% RSLogix 500 project CTD QUE 3.RSS, saved by version 8.30.00.15 %
PROJECT "UNTITLED"    % processor: MicroLogix 1400 %

PROGRAM FILES
  LAD 2   6 rungs

DATA FILES
  O0 OUTPUT  6 elements
  I1 INPUT  8 elements
  S2 STATUS  66 elements
  B3 BINARY  1 elements
  T4 TIMER  1 elements
  C5 COUNTER  6 elements
  R6 CONTROL  1 elements
  N7 INTEGER  1 elements
  F8 FLOAT  1 elements

LADDER 2
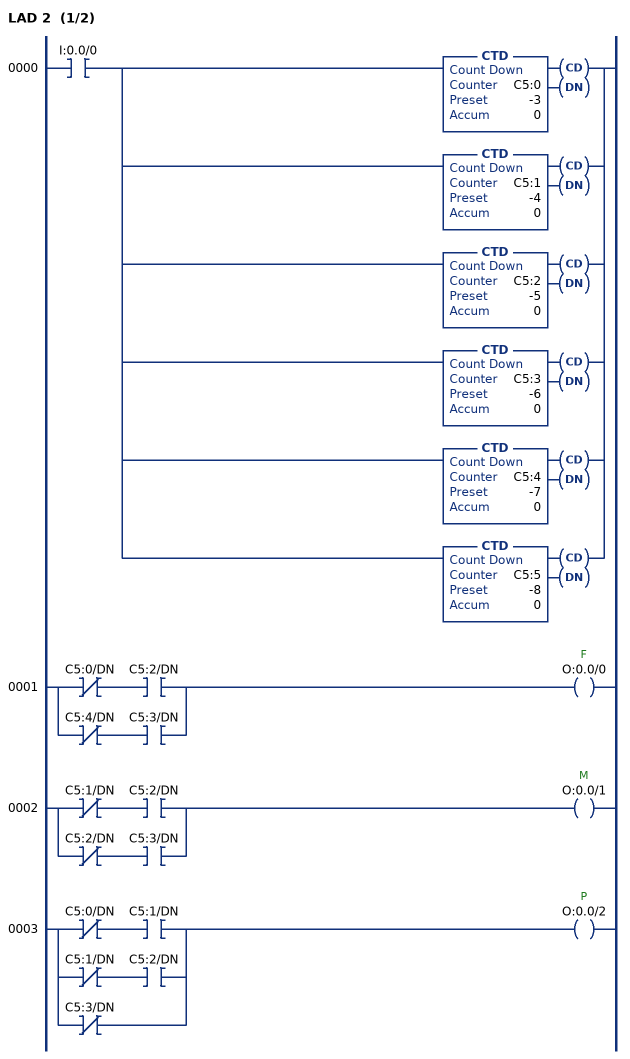
% Rung: 0 %  % edit flag set %
SOR XIC I:0.0/0 BST CTD C5:0 -3 0 NXB BST CTD C5:1 -4 0 NXB BST CTD C5:2 -5 0 NXB BST CTD C5:3 -6 0 NXB BST CTD C5:4 -7 0 NXB CTD C5:5 -8 0 BND BND BND BND BND EOR
% Rung: 1 %
SOR BST XIO C5:0/DN XIC C5:2/DN NXB XIO C5:4/DN XIC C5:3/DN BND OTE O:0.0/0 EOR
%   O:0.0/0  F %
% Rung: 2 %
SOR BST XIO C5:1/DN XIC C5:2/DN NXB XIO C5:2/DN XIC C5:3/DN BND OTE O:0.0/1 EOR
%   O:0.0/1  M %
% Rung: 3 %
SOR BST XIO C5:0/DN XIC C5:1/DN NXB BST XIO C5:1/DN XIC C5:2/DN NXB XIO C5:3/DN BND BND OTE O:0.0/2 EOR
%   O:0.0/2  P %

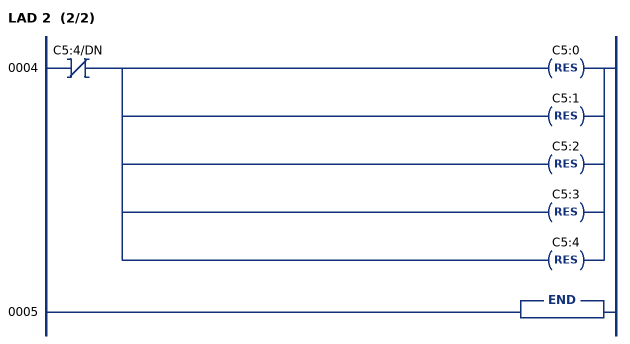
% Rung: 4 %
SOR XIO C5:4/DN BST RES C5:0 NXB BST RES C5:1 NXB BST RES C5:2 NXB BST RES C5:3 NXB RES C5:4 BND BND BND BND EOR
% Rung: 5 %
SOR END EOR

DATA TABLE (non-zero values as saved)
DATA C5
% .PRE .ACC %
% C5:0 % -3 0
% C5:1 % -4 0
% C5:2 % -5 0
% C5:3 % -6 0
% C5:4 % -7 0
% C5:5 % -8 0
